FUNCTION_BLOCK EL3453
VAR
	_io : EL3453_Data;
	{attribute addProperty Name "WcState"}
	_wcState : WcStateInputToggle;
	{attribute addProperty Name "Info data"}
	_infoData : InfoDataAds;
END_VAR

PROPERTY IO : REFERENCE TO EL3453_Data
GET
IO REF= _io;
END_GET
END_PROPERTY

PROPERTY WcState : REFERENCE TO WcStateInputToggle
GET
WcState REF= _wcState;
END_GET
END_PROPERTY

END_FUNCTION_BLOCK

(* stored: Version 1.1.0.1, ProductVersion 3.1.4024.9
   POU EL3453: Id {fc8fc785-be11-0ad3-27d3-b3ab02168737}, SpecialFunc None
   Property IO: Id {2dd1f1ca-e776-0c8a-1288-0670e78c07ba}
   Get Get: Id {683d7bbe-f26a-02dd-38e8-c0c9895e54d7}
   Property WcState: Id {2927ce4b-5a88-061b-1c61-168a14cc281b}
   Get Get: Id {97b88493-2998-024b-2b33-7b5036589eea} *)
